INTERFACE ITF_TopElement_HMI_Connector EXTENDS ITF_BaseTopElement_HMI_Connector

END_INTERFACE

(* stored: Version 1.1.0.1, ProductVersion 3.1.4024.15
   Itf ITF_TopElement_HMI_Connector: Id {0f399b32-572b-4586-8360-47530c3a45ce} *)
